TYPE ST_APP_INFO :
STRUCT
  AppInit           : E_PROGRESS;
  Instance          : E_INSTANCE;  // process ID from which the MoverPerMinute counter is copied
  MoverPerMinute    : UDINT;
  MoverTotal        : UDINT;
  StationParameterVariant : UDINT;
END_STRUCT
END_TYPE

(* stored: Version 1.1.0.1, ProductVersion 3.1.4026.20
   DUT ST_APP_INFO: Id {a76488ed-38c5-4433-84c6-4d201239df77} *)
